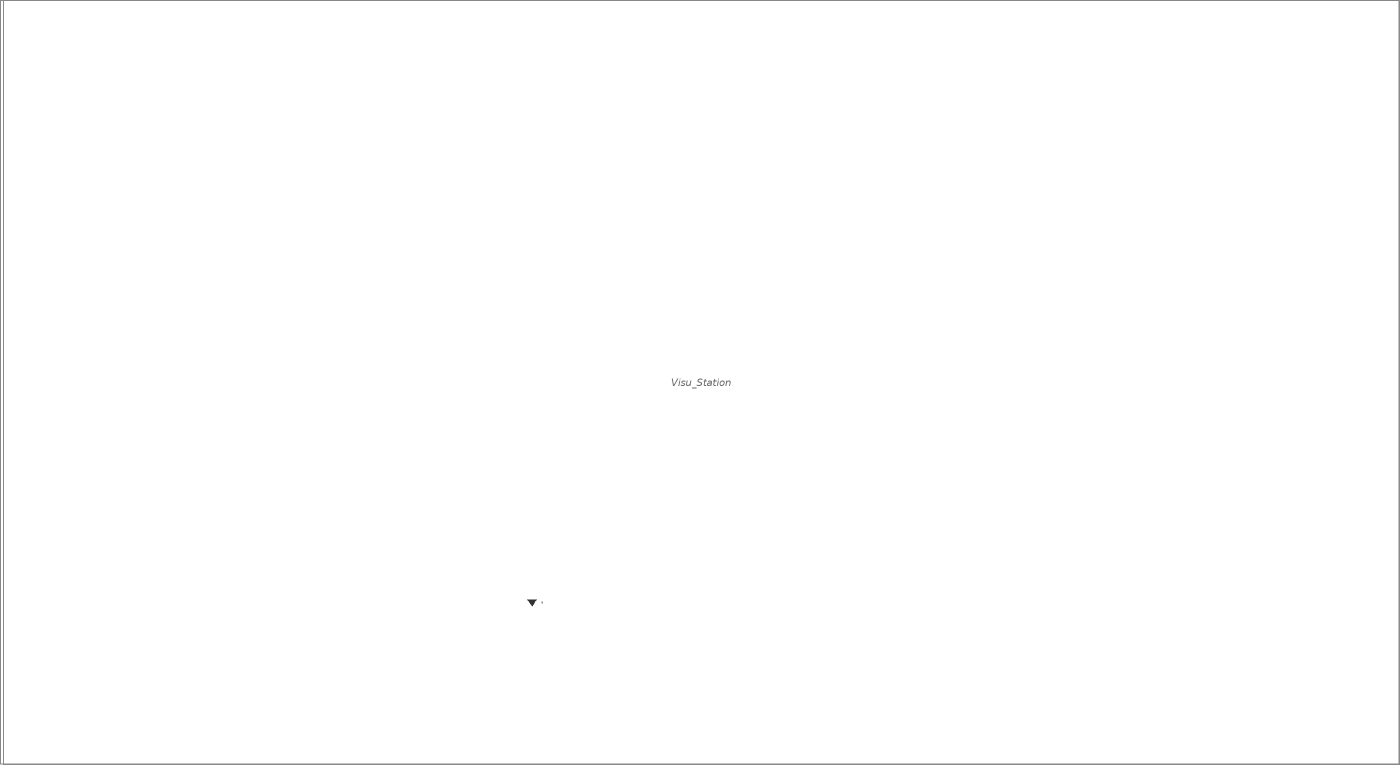
VISUALIZATION Main_Visu  // 1453x794
    SpinControl (562,625 1x0)
    TabControl (3,0 1450x794)
        shows Visu_Station(fbStation := MAIN.fbStation01)
        shows Visu_Station(fbStation := MAIN.fbStation02)
        [0]: TabTitle=ChargingStation01
        [1]: TabTitle=ChargingStation02
END_VISUALIZATION

(* stored: Version 1.1.0.1
   Visu Main_Visu: Id {286bfbd1-e8d1-4ab6-86aa-344f7e32fee8} *)
